{attribute 'pack_mode' := '1'}
TYPE ChangeAxisEnable EXTENDS IncomingMessage :
STRUCT
	axisIndex: DINT; (* 1 or 2.*)
	enabled: BOOL;
END_STRUCT
END_TYPE

(* stored: Version 1.1.0.1, ProductVersion 3.1.4022.12
   DUT ChangeAxisEnable: Id {7211e326-19e7-4ff0-a147-32508ee40742} *)
